FUNCTION_BLOCK EM_OutfeedA EXTENDS FB_Transport
VAR

END_VAR

END_FUNCTION_BLOCK

(* stored: Version 1.1.0.1, ProductVersion 3.1.4024.12
   POU EM_OutfeedA: Id {2864aa0f-79f4-4c15-96e2-8d7a37ae349b}, SpecialFunc None *)
